(*
SPDX-FileCopyrightText: Â© 2026 Oleksandr Tiutyk <trofimich@gmail.com>
SPDX-License-Identifier: MIT
License: https://opensource.org/license/mit
*)

(*!
<summary>Base converter providing linear interpolation and boundary clamping
between raw and engineering values.</summary>
<description>
Maps an input value proportionally between configured minimum and maximum limits.
Clamps values outside range to boundary limits and defends against division by zero.
For a range with distinct engineering limits and equal raw limits, output conversion returns the common raw limit.
</description>
*)

{attribute 'no_explicit_call' := 'do not call this function block directly'}
FUNCTION_BLOCK ABSTRACT AbstractRangeAnalogValueConverter EXTENDS TOF_Core.Object IMPLEMENTS IAnalogValueConverter
VAR
	{attribute 'hide'} 
	_MinAnalogValue : REFERENCE TO LREAL;
	{attribute 'hide'} 
	_MaxAnalogValue : REFERENCE TO LREAL;
	{attribute 'hide'} 
	_MinRawValue : REFERENCE TO RAW_ANALOG_VALUE;
	{attribute 'hide'} 
	_MaxRawValue : REFERENCE TO RAW_ANALOG_VALUE;
END_VAR

(*!
<summary>Converts an engineering unit value to raw hardware representation with boundary clamping.</summary>
<description>
If the engineering limits differ and the raw limits are equal, returns the common limit in the requested
raw representation. An INT16 result has zeroed upper bytes.
</description>
<param name="analogValue">Engineering unit analog value.</param>
<param name="rawValueType">Target raw data representation.</param>
*)
METHOD ConvertAnalogValueToRawValue : RAW_ANALOG_VALUE
VAR_INPUT
	analogValue	: LREAL;
	rawValueType : RAW_ANALOG_VALUE_TYPE;
END_VAR
VAR
	formattedExceptionMessage : TOF_Core.ERROR_MESSAGE;

	minRawValueLReal : LREAL;
	maxRawValueLReal : LREAL;
	rawValueLReal : LREAL;
	
	exceptionCode : __SYSTEM.ExceptionCode;	
END_VAR
IF NOT __ISVALIDREF(_MinAnalogValue)
	OR_ELSE NOT __ISVALIDREF(_MaxAnalogValue)
	OR_ELSE NOT __ISVALIDREF(_MinRawValue)
	OR_ELSE NOT __ISVALIDREF(_MaxRawValue)
	OR_ELSE _MinAnalogValue = _MaxAnalogValue
THEN
	RETURN;
END_IF

IF _MaxAnalogValue > _MinAnalogValue THEN
	IF analogValue >= _MaxAnalogValue THEN
		analogValue := _MaxAnalogValue;
	ELSIF analogValue <= _MinAnalogValue THEN
		analogValue := _MinAnalogValue;
	END_IF
ELSIF _MaxAnalogValue < _MinAnalogValue THEN
	IF analogValue <= _MaxAnalogValue THEN
		analogValue := _MaxAnalogValue;
	ELSIF analogValue >= _MinAnalogValue THEN
		analogValue := _MinAnalogValue;
	END_IF
END_IF

CASE rawValueType OF
	RAW_ANALOG_VALUE_TYPE.INT16:
		minRawValueLReal := TO_LREAL(_MinRawValue.Int16);
		maxRawValueLReal := TO_LREAL(_MaxRawValue.Int16);

	RAW_ANALOG_VALUE_TYPE.INT32:
		minRawValueLReal := TO_LREAL(_MinRawValue.Int32);
		maxRawValueLReal := TO_LREAL(_MaxRawValue.Int32);

	RAW_ANALOG_VALUE_TYPE.REAL32:
		minRawValueLReal := TO_LREAL(_MinRawValue.Real32);
		maxRawValueLReal := TO_LREAL(_MaxRawValue.Real32);

	ELSE
		RETURN;
END_CASE

IF minRawValueLReal = maxRawValueLReal THEN
	CASE rawValueType OF
		RAW_ANALOG_VALUE_TYPE.INT16:
			ConvertAnalogValueToRawValue := RawAnalogValues.FromInt16(value := _MinRawValue.Int16);

		RAW_ANALOG_VALUE_TYPE.INT32:
			ConvertAnalogValueToRawValue := RawAnalogValues.FromInt32(value := _MinRawValue.Int32);

		RAW_ANALOG_VALUE_TYPE.REAL32:
			ConvertAnalogValueToRawValue := RawAnalogValues.FromReal32(value := _MinRawValue.Real32);
	END_CASE

	RETURN;
END_IF

__TRY
	rawValueLReal := (analogValue - _MinAnalogValue) / (_MaxAnalogValue - _MinAnalogValue)
		* (maxRawValueLReal - minRawValueLReal) + minRawValueLReal;
__CATCH(exceptionCode)
	formattedExceptionMessage := TOF_Core.WideStrings.Concat255(
		"Invalid analog to raw value conversion. Exception code: ",
		TO_WSTRING(exceptionCode)
	);

	TOF_Core.Exceptions.ThrowStandard(
		sourceNamespaceName := NamespaceName,
		sourceClassName := ClassName,
		sourcePOUName := __POUNAME(),
		sourcePosition := __POSITION(),
		message := formattedExceptionMessage
	);
__ENDTRY

ConvertAnalogValueToRawValue.Int32 := 0;

CASE rawValueType OF
	RAW_ANALOG_VALUE_TYPE.INT16:
		ConvertAnalogValueToRawValue.Int16 := TO_INT(rawValueLReal);

	RAW_ANALOG_VALUE_TYPE.INT32:
		ConvertAnalogValueToRawValue.Int32 := TO_DINT(rawValueLReal);

	RAW_ANALOG_VALUE_TYPE.REAL32:
		ConvertAnalogValueToRawValue.Real32 := TO_REAL(rawValueLReal);
END_CASE
END_METHOD

(*!
<summary>Converts raw hardware representation to an engineering unit value with boundary clamping.</summary>
<param name="rawValue">Raw process value union.</param>
<param name="rawValueType">Source raw data representation.</param>
*)
METHOD ConvertRawValueToAnalogValue : LREAL
VAR_INPUT
	rawValue : RAW_ANALOG_VALUE;
	rawValueType : RAW_ANALOG_VALUE_TYPE;
END_VAR
VAR
	formattedExceptionMessage : TOF_Core.ERROR_MESSAGE;

	rawValueLReal : LREAL;
	minRawValueLReal : LREAL;
	maxRawValueLReal : LREAL;

	exceptionCode : __SYSTEM.ExceptionCode;
END_VAR
IF NOT __ISVALIDREF(_MinAnalogValue)
	OR_ELSE NOT __ISVALIDREF(_MaxAnalogValue)
	OR_ELSE NOT __ISVALIDREF(_MinRawValue)
	OR_ELSE NOT __ISVALIDREF(_MaxRawValue)
	OR_ELSE _MinAnalogValue = _MaxAnalogValue
THEN
	RETURN;
END_IF

CASE rawValueType OF
	RAW_ANALOG_VALUE_TYPE.INT16:
		rawValueLReal := TO_LREAL(rawValue.Int16);
		minRawValueLReal := TO_LREAL(_MinRawValue.Int16);
		maxRawValueLReal := TO_LREAL(_MaxRawValue.Int16);

	RAW_ANALOG_VALUE_TYPE.INT32:
		rawValueLReal := TO_LREAL(rawValue.Int32);
		minRawValueLReal := TO_LREAL(_MinRawValue.Int32);
		maxRawValueLReal := TO_LREAL(_MaxRawValue.Int32);

	RAW_ANALOG_VALUE_TYPE.REAL32:
		rawValueLReal := TO_LREAL(rawValue.Real32);
		minRawValueLReal := TO_LREAL(_MinRawValue.Real32);
		maxRawValueLReal := TO_LREAL(_MaxRawValue.Real32);

	ELSE
		RETURN;
END_CASE

IF maxRawValueLReal > minRawValueLReal THEN
	IF rawValueLReal >= maxRawValueLReal THEN
		ConvertRawValueToAnalogValue := _MaxAnalogValue;
		RETURN;
	ELSIF rawValueLReal <= minRawValueLReal THEN
		ConvertRawValueToAnalogValue := _MinAnalogValue;
		RETURN;
	END_IF
ELSIF maxRawValueLReal < minRawValueLReal THEN
	IF rawValueLReal <= maxRawValueLReal THEN
		ConvertRawValueToAnalogValue := _MaxAnalogValue;
		RETURN;
	ELSIF rawValueLReal >= minRawValueLReal THEN
		ConvertRawValueToAnalogValue := _MinAnalogValue;
		RETURN;
	END_IF
ELSE
	ConvertRawValueToAnalogValue := _MinAnalogValue;
	RETURN;
END_IF

__TRY
	ConvertRawValueToAnalogValue := (rawValueLReal - minRawValueLReal) / (maxRawValueLReal - minRawValueLReal)
		* (_MaxAnalogValue - _MinAnalogValue) + _MinAnalogValue;
__CATCH(exceptionCode)
	formattedExceptionMessage := TOF_Core.WideStrings.Concat255(
		"Invalid raw to analog value conversion. Exception code: ",
		TO_WSTRING(exceptionCode)
	);

	TOF_Core.Exceptions.ThrowStandard(
		sourceNamespaceName := NamespaceName,
		sourceClassName := ClassName,
		sourcePOUName := __POUNAME(),
		sourcePosition := __POSITION(),
		message := formattedExceptionMessage
	);
__ENDTRY
END_METHOD

(*!
<summary>Gets a reference to the maximum engineering unit value.</summary>
*)
{attribute 'monitoring' := 'call'}
PROPERTY FINAL MaxAnalogValue : REFERENCE TO LREAL
GET
MaxAnalogValue REF= _MaxAnalogValue;
END_GET
END_PROPERTY

(*!
<summary>Gets a reference to the maximum raw process value.</summary>
*)
{attribute 'monitoring' := 'call'}
PROPERTY FINAL MaxRawValue : REFERENCE TO RAW_ANALOG_VALUE
GET
MaxRawValue REF= _MaxRawValue;
END_GET
END_PROPERTY

(*!
<summary>Gets a reference to the minimum engineering unit value.</summary>
*)
{attribute 'monitoring' := 'call'}
PROPERTY FINAL MinAnalogValue : REFERENCE TO LREAL
GET
MinAnalogValue REF= _MinAnalogValue;
END_GET
END_PROPERTY

(*!
<summary>Gets a reference to the minimum raw process value.</summary>
*)
{attribute 'monitoring' := 'call'}
PROPERTY FINAL MinRawValue : REFERENCE TO RAW_ANALOG_VALUE
GET
MinRawValue REF= _MinRawValue;
END_GET
END_PROPERTY

(*!
<summary>Gets the namespace name of the converter.</summary>
*)
{attribute 'monitoring' := 'call'}
PROPERTY NamespaceName : REFERENCE TO STRING
GET
NamespaceName REF= CurrentNamespace.Name;
END_GET
END_PROPERTY

END_FUNCTION_BLOCK

(* stored: Version 1.1.0.1
   POU AbstractRangeAnalogValueConverter: Id {c2526683-36df-499d-8472-588820322f0f}, SpecialFunc None
   Method ConvertAnalogValueToRawValue: Id {baf39a83-01bf-44c2-8637-07e8713fb214}
   Method ConvertRawValueToAnalogValue: Id {2b018a58-1ace-42e8-a492-2c6a67a392cf}
   Property MaxAnalogValue: Id {a941654f-d717-4440-bc44-ed518a303456}
   Get Get: Id {d8c2c8ae-ba7a-4f28-828a-6d7d272b4399}
   Property MaxRawValue: Id {3b0fa350-39b1-4e9e-bd2f-9c6f49af8305}
   Get Get: Id {7cef5b0c-1235-4d8f-a4b6-b6fb9a494744}
   Property MinAnalogValue: Id {c1129997-b2c7-4985-a7e1-2c2a53b652a2}
   Get Get: Id {ba9e5b85-6e7d-4f21-8e43-68be353a5dfe}
   Property MinRawValue: Id {fc2912d7-e9eb-424a-a71c-e00912e1679a}
   Get Get: Id {0bac5199-db63-4ede-964c-b45620359765}
   Property NamespaceName: Id {4ac53464-c80d-49f6-9468-789d3c010411}
   Get Get: Id {af413a5a-e5d5-41cd-8275-68368a979eb9} *)
